Staubli VAL3: onF7Event.pgx

program onF7Event(bool& x_bSave[])
  local mdesc l_mDesc
  local num l_nMoveType
  local bool l_bStop
  local num l_nTcpAction
  local num l_nItem
  local string l_sEmpty
  local num l_nDone
  local num l_nStop
begin
//  // look if the bButton is enable
//  if bButton[6]
//    //
//    // insert the user one
//    l_nItem=nIndex
//    call trajType:insertItem(nIndex,nIndex+1)
//    // empty one
//    l_sEmpty=""
//    l_bStop=false
//    l_nDone=0
//    call trajType:getTrajItem(l_tTraj,nIndex)
//    call trajType:setTrajItem(l_tTraj,nIndex+1)
//    x_bSave=true
//    nSelect=nSelect+1
//  endIf
end
